// TIA Portal V15 export
// export: Created 2018-05-30T14:06:05.1178745Z, ExportSetting WithDefaults, WithReadOnly, DisplayName Totally Integrated Automation Portal, DisplayVersion V15, DisplayName STEP 7 Professional, DisplayVersion V15, DisplayName WinCC Professional, DisplayVersion V15, DisplayName TIA Portal Openness, DisplayVersion V15
FUNCTION_BLOCK "BST_MOTOR_400"   // FB21, STL
{ S7_Optimized_Access := 'FALSE' }
VERSION : 0.1
// stored: AutoNumber false, CodeModifiedDate 2018-05-30T13:59:14.5053889Z, CompileDate 2018-05-30T13:59:14.5053888Z, CreationDate 2018-05-30T13:55:26.8283664Z, InterfaceModifiedDate 2018-05-30T13:59:03.2547453Z, IsConsistent true, IsKnowHowProtected false, ISMultiInstanceCapable true, IsWriteProtected false, LibraryConformanceStatus The object is library-conformant., ModifiedDate 2018-05-30T13:59:14.5053889Z, ParameterModified 2018-05-30T13:59:03.2547453Z, StructureModified 2018-05-30T13:59:03.2547453Z, UDAEnableTagReadback false
   VAR_INPUT
      AUTO_ON : Bool;
      L_AUT : Bool;
      FB_ON : Bool;
      ERR_EXTERN : Bool;
   END_VAR
   VAR_OUTPUT
      QRUN : Bool;
      QSTOP : Bool;
      QCMD_ON : Bool;
      QMON_ERR : Bool;
      QMPS : Bool;
      QERR : Bool;
   END_VAR
BEGIN
END_FUNCTION_BLOCK
